FUNCTION_BLOCK SF_ResetButton (* PLCopen Safety SF_ResetButton (Part 1 v2.10, Ch. 6.1) - Trailing-Edge Reset *)
  (* Standard: 61499-2; Function: Adds Trailing-Edge functionality (LOW-HIGH-LOW) to Reset inputs, per EN ISO 13849-1:2015 5.2.2. ResetOut pulses TRUE for 1 cycle after a valid press-and-release within [TrailingMinimum, TrailingMaximum].; Description: Copyright (c) 2026 Meisterschulen am Ostbahnhof This program and the accompanying materials are made available under the terms of the Eclipse Public License 2.0 which is available at https://www.eclipse.org/legal/epl-2.0/ SPDX-License-Identifier: EPL-2.0 *)
  (* Version 1.0, 2026-10-09, Franz Höpfinger, Meisterschulen am Ostbahnhof, Modeled after logiBUS::utils::sequence::timed::sequence_T_05 (ECC + ATimeOut Plug pattern). Source: PLCopen TC5 Safety Part 1 - Concepts and Function Blocks, Version 2.10, Nov. 7 2023, Chapter 6.1 Reset Button. *)
  PACKAGE logiBUS::safety::PLCopen;
  IMPORT logiBUS::safety::PLCopen::const::DiagCodes;
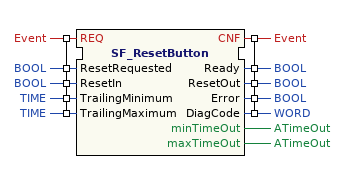
  EVENT_INPUT
    REQ WITH ResetRequested, ResetIn, TrailingMinimum, TrailingMaximum; (* Cyclic evaluation request *)
  END_EVENT
  EVENT_OUTPUT
    CNF WITH Ready, ResetOut, Error, DiagCode; (* Confirmation of Requested Service *)
  END_EVENT
  VAR_INPUT
    ResetRequested : BOOL := TRUE; (* From the paired FB's ResetRequest output. TRUE=monitor ResetIn, FALSE=inactive *)
    ResetIn : BOOL := FALSE; (* Reset button input. FALSE=released, TRUE=actuated *)
    TrailingMinimum : TIME := T#350ms; (* Min. actuation time (absolute min 100ms). Shorter presses are ignored *)
    TrailingMaximum : TIME := T#2s; (* Max. actuation time. Longer presses are ignored *)
  END_VAR
  VAR_OUTPUT
    Ready : BOOL := FALSE; (* FB active, outputs valid *)
    ResetOut : BOOL := FALSE; (* 1-cycle pulse: valid trailing-edge reset detected *)
    Error : BOOL := FALSE; (* TRUE while in an error state, see DiagCode *)
    DiagCode : WORD := 16#0000; (* FB-specific status/error code, see PLCopen Safety Part 1 Ch. 6.1.6 *)
  END_VAR
  PLUGS
    minTimeOut : iec61499::events::ATimeOut; (* TrailingMinimum timer *)
    maxTimeOut : iec61499::events::ATimeOut; (* TrailingMaximum timer *)
  END_PLUGS
  VAR
    xPrevResetIn : BOOL := FALSE; (* ResetIn value as of the previous scan, for edge detection *)
    xMinOk : BOOL := FALSE; (* Latched TRUE once TrailingMinimum has elapsed since the rising edge *)
    xParamOk : BOOL := FALSE; (* TrailingMinimum/TrailingMaximum are within the valid range *)
  END_VAR
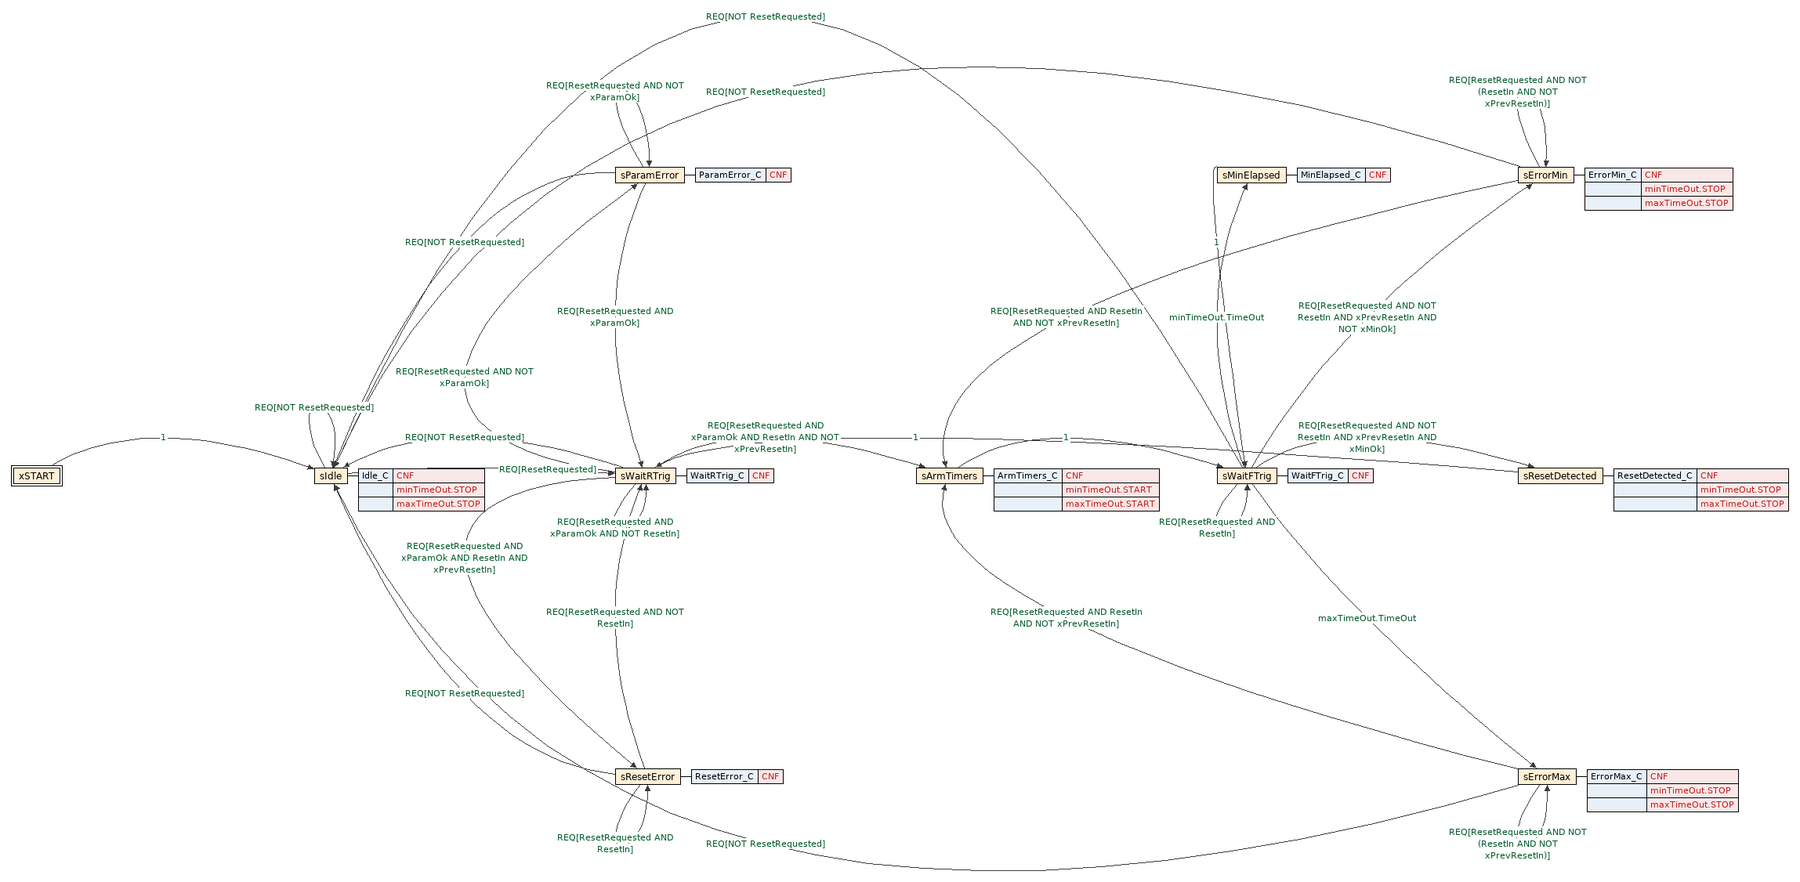
  EC_STATES
    xSTART; (* Initial State *)
    sIdle : Idle_C -> CNF, -> minTimeOut.STOP, -> maxTimeOut.STOP;
    sParamError : ParamError_C -> CNF;
    sResetError : ResetError_C -> CNF;
    sWaitRTrig : WaitRTrig_C -> CNF;
    sArmTimers : ArmTimers_C -> CNF, -> minTimeOut.START, -> maxTimeOut.START; (* One-shot: (re)start both timers, then fall through to sWaitFTrig *)
    sWaitFTrig : WaitFTrig_C -> CNF;
    sMinElapsed : MinElapsed_C -> CNF; (* One-shot: latch xMinOk, then fall through back to sWaitFTrig *)
    sErrorMin : ErrorMin_C -> CNF, -> minTimeOut.STOP, -> maxTimeOut.STOP;
    sErrorMax : ErrorMax_C -> CNF, -> minTimeOut.STOP, -> maxTimeOut.STOP;
    sResetDetected : ResetDetected_C -> CNF, -> minTimeOut.STOP, -> maxTimeOut.STOP;
  END_STATES
  EC_TRANSITIONS
    xSTART TO sIdle := 1;
    sIdle TO sIdle := REQ[NOT ResetRequested];
    sIdle TO sWaitRTrig := REQ[ResetRequested];
    sParamError TO sIdle := REQ[NOT ResetRequested];
    sParamError TO sParamError := REQ[ResetRequested AND NOT xParamOk];
    sParamError TO sWaitRTrig := REQ[ResetRequested AND xParamOk];
    sResetError TO sIdle := REQ[NOT ResetRequested];
    sResetError TO sResetError := REQ[ResetRequested AND ResetIn];
    sResetError TO sWaitRTrig := REQ[ResetRequested AND NOT ResetIn];
    sWaitRTrig TO sIdle := REQ[NOT ResetRequested];
    sWaitRTrig TO sParamError := REQ[ResetRequested AND NOT xParamOk];
    sWaitRTrig TO sResetError := REQ[ResetRequested AND xParamOk AND ResetIn AND xPrevResetIn];
    sWaitRTrig TO sArmTimers := REQ[ResetRequested AND xParamOk AND ResetIn AND NOT xPrevResetIn];
    sWaitRTrig TO sWaitRTrig := REQ[ResetRequested AND xParamOk AND NOT ResetIn];
    sArmTimers TO sWaitFTrig := 1;
    sWaitFTrig TO sIdle := REQ[NOT ResetRequested];
    sWaitFTrig TO sResetDetected := REQ[ResetRequested AND NOT ResetIn AND xPrevResetIn AND xMinOk];
    sWaitFTrig TO sErrorMin := REQ[ResetRequested AND NOT ResetIn AND xPrevResetIn AND NOT xMinOk];
    sWaitFTrig TO sWaitFTrig := REQ[ResetRequested AND ResetIn];
    sWaitFTrig TO sMinElapsed := minTimeOut.TimeOut;
    sWaitFTrig TO sErrorMax := maxTimeOut.TimeOut;
    sMinElapsed TO sWaitFTrig := 1;
    sErrorMin TO sIdle := REQ[NOT ResetRequested];
    sErrorMin TO sArmTimers := REQ[ResetRequested AND ResetIn AND NOT xPrevResetIn];
    sErrorMin TO sErrorMin := REQ[ResetRequested AND NOT (ResetIn AND NOT xPrevResetIn)];
    sErrorMax TO sIdle := REQ[NOT ResetRequested];
    sErrorMax TO sArmTimers := REQ[ResetRequested AND ResetIn AND NOT xPrevResetIn];
    sErrorMax TO sErrorMax := REQ[ResetRequested AND NOT (ResetIn AND NOT xPrevResetIn)];
    sResetDetected TO sWaitRTrig := 1;
  END_TRANSITIONS
  ALGORITHM Idle_C IN ST:
 // 0000 Idle - FB not active
xParamOk := (TrailingMinimum <= TrailingMaximum) AND (TrailingMinimum >= T#100ms);
Ready := BOOL#FALSE;
ResetOut := BOOL#FALSE;
Error := BOOL#FALSE;
DiagCode := DiagCodes::IDLE;
xPrevResetIn := ResetIn;
  END_ALGORITHM
  ALGORITHM ParamError_C IN ST:
 // C000 Parameter Error - TrailingMinimum > TrailingMaximum OR TrailingMinimum < 100ms
xParamOk := (TrailingMinimum <= TrailingMaximum) AND (TrailingMinimum >= T#100ms);
Ready := BOOL#TRUE;
ResetOut := BOOL#FALSE;
Error := BOOL#TRUE;
DiagCode := DiagCodes::PARAMETER_ERROR;
xPrevResetIn := ResetIn;
  END_ALGORITHM
  ALGORITHM ResetError_C IN ST:
 // C001 Reset Error - ResetIn was already TRUE when ResetRequested became TRUE
Ready := BOOL#TRUE;
ResetOut := BOOL#FALSE;
Error := BOOL#TRUE;
DiagCode := DiagCodes::RESET_ERROR;
xPrevResetIn := ResetIn;
  END_ALGORITHM
  ALGORITHM WaitRTrig_C IN ST:
 // 83E2 Wait for R_TRIG - enabled, waiting for the operator to press the button
Ready := BOOL#TRUE;
ResetOut := BOOL#FALSE;
Error := BOOL#FALSE;
DiagCode := DiagCodes::WAIT_R_TRIG;
xPrevResetIn := ResetIn;
  END_ALGORITHM
  ALGORITHM ArmTimers_C IN ST:
 // 83F2 (entry) - rising edge detected, (re)start both trailing-edge timers
minTimeOut.DT := TrailingMinimum;
maxTimeOut.DT := TrailingMaximum;
xMinOk := BOOL#FALSE;
Ready := BOOL#TRUE;
ResetOut := BOOL#FALSE;
Error := BOOL#FALSE;
DiagCode := DiagCodes::WAIT_F_TRIG;
xPrevResetIn := ResetIn;
  END_ALGORITHM
  ALGORITHM WaitFTrig_C IN ST:
 // 83F2 Wait for F_TRIG - ResetIn is TRUE, waiting for release
Ready := BOOL#TRUE;
ResetOut := BOOL#FALSE;
Error := BOOL#FALSE;
DiagCode := DiagCodes::WAIT_F_TRIG;
xPrevResetIn := ResetIn;
  END_ALGORITHM
  ALGORITHM MinElapsed_C IN ST:
 // TrailingMinimum elapsed while still waiting for F_TRIG - latch it, state stays 83F2
xMinOk := BOOL#TRUE;
Ready := BOOL#TRUE;
ResetOut := BOOL#FALSE;
Error := BOOL#FALSE;
DiagCode := DiagCodes::WAIT_F_TRIG;
  END_ALGORITHM
  ALGORITHM ErrorMin_C IN ST:
 // C3F0 Error Trailing Minimum - F_TRIG before TrailingMinimum elapsed. Waiting for R_TRIG
Ready := BOOL#TRUE;
ResetOut := BOOL#FALSE;
Error := BOOL#TRUE;
DiagCode := DiagCodes::ERROR_TRAILING_MINIMUM;
xPrevResetIn := ResetIn;
  END_ALGORITHM
  ALGORITHM ErrorMax_C IN ST:
 // C3E0 Error Trailing Maximum - TrailingMaximum elapsed before F_TRIG. Waiting for R_TRIG
Ready := BOOL#TRUE;
ResetOut := BOOL#FALSE;
Error := BOOL#TRUE;
DiagCode := DiagCodes::ERROR_TRAILING_MAXIMUM;
xPrevResetIn := ResetIn;
  END_ALGORITHM
  ALGORITHM ResetDetected_C IN ST:
 // 8000 Reset Detected - valid trailing-edge reset, 1-cycle pulse on ResetOut
Ready := BOOL#TRUE;
ResetOut := BOOL#TRUE;
Error := BOOL#FALSE;
DiagCode := DiagCodes::RESET_DETECTED;
xPrevResetIn := ResetIn;
  END_ALGORITHM
END_FUNCTION_BLOCK
(* other elements stored in the file *)
(* Fig. 15 branches "Wait for R_TRIG" into: bad params (0), stuck ResetIn without a fresh edge (1), a fresh rising edge (2, -> sArmTimers/sWaitFTrig), else self-loop. *)
